(* CODESYS project PETO.export

Project tree, tasks and I/O mapping:
  Device : CODESYS Control Win V3 x64, CODESYS, version 3.5.21.40
    application Application
      libraries: Standard, 3.5.18.0 (System); Util, 3.5.21.0 (System)
      task AlarmManagerTask (cyclic, interval 50 ms, priority 31) calls AlarmManager.Alarm_Prg
      task MainTask (cyclic, interval t#20ms, priority 1) calls COMPROBACION, PREPARACION, SERVIR, SALIDAS
      task VISU_TASK (cyclic, interval 100 ms, priority 31) calls VisuElems.Visu_Prg
      Alarm Configuration
        alarm class Error (priority 10, acknowledge ACK)
        alarm class Info (priority 100, acknowledge REP)
        alarm class Warning (priority 30, acknowledge REP)
        alarm group AlarmGroup
            0 [Error]: Comparison Equal, ExpressionToCompare TRUE, Expression PREPARACION.ErrC - "Falla en el calentador"
            1 [Error]: Comparison Equal, ExpressionToCompare TRUE, Expression PREPARACION.ErrM - "Falla del motor mezclador"
        AlarmStorage
        text list AlarmGroup
      program COMPROBACION [LD]
      visualisation Visualization
  program PREPARACION [LD]
  program SALIDAS [LD]
  program SERVIR [LD]
*)

// Device/Application/COMPROBACION
PROGRAM COMPROBACION
VAR
	START: BOOL;
	STOP: BOOL;
	Inicio: BOOL;
	VO: BOOL;
	Current_State: INT := 10;
	State_machine: INT := 10;
	P1: BOOL;
	L1: BOOL;
	Q1: BOOL;
	RE: BOOL;
	D: BOOL;
	aux1: BOOL;
	V: BOOL;
	aux2: BOOL;
END_VAR
VAR // added by the converter: edge detectors and wires of the graphical bodies
    _w1, _w2, _w3 : BOOL;
END_VAR

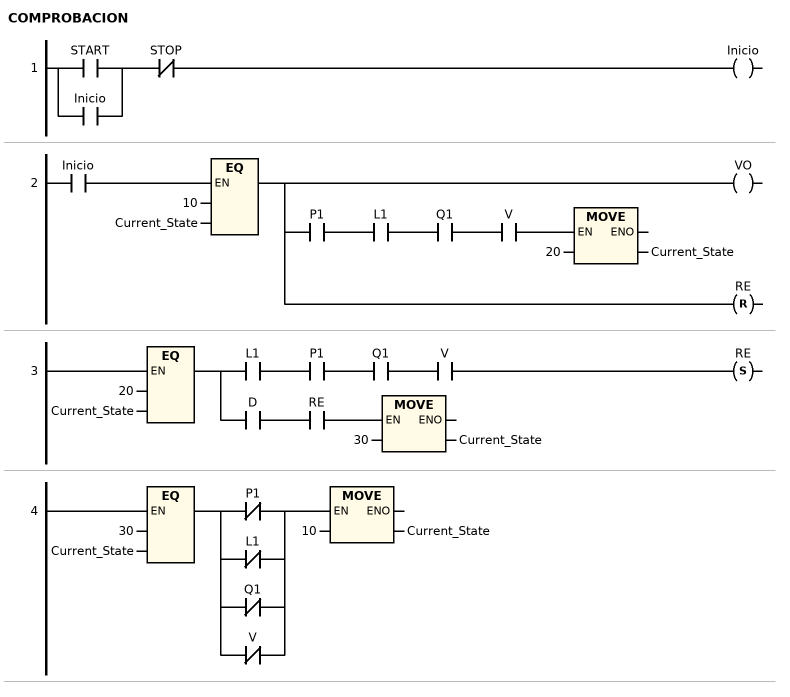
// NETWORK 1
Inicio := (START OR Inicio) AND NOT STOP;

// NETWORK 2
_w1 := Inicio AND 10 = Current_State;
VO := _w1;
IF _w1 AND P1 AND L1 AND Q1 AND V THEN Current_State := 20; END_IF
RE R= _w1;

// NETWORK 3
_w2 := 20 = Current_State;
RE S= _w2 AND L1 AND P1 AND Q1 AND V;
IF _w2 AND D AND RE THEN Current_State := 30; END_IF

// NETWORK 4
_w3 := 30 = Current_State;
IF _w3 AND (NOT P1 OR NOT L1 OR NOT Q1 OR NOT V) THEN Current_State := 10; END_IF

END_PROGRAM

// PREPARACION
PROGRAM PREPARACION
VAR
	RE: BOOL;
	aux1: BOOL;
	CCurrent_State: INT := 10;
	P2: BOOL;
	M1: BOOL;
	// Calentadaor
	K1: BOOL;
	// motor principal
	MO: BOOL;
	TIMERPETO: TON;
	// el tiempo de espera se cumplio
	Tim1: BOOL;
	// error de calentador
	ErrC: BOOL;
	// temperatura tanque
	H1: INT;
	// MANTENIMIENTO
	Mt: BOOL;
	// error de motor
	ErrM: BOOL;
	TIMERMOTOR: TON;
	// peto listo
	Ro: BOOL;
END_VAR
VAR // added by the converter: edge detectors and wires of the graphical bodies
    _w1, _w2, _w3, _w4 : BOOL;
END_VAR

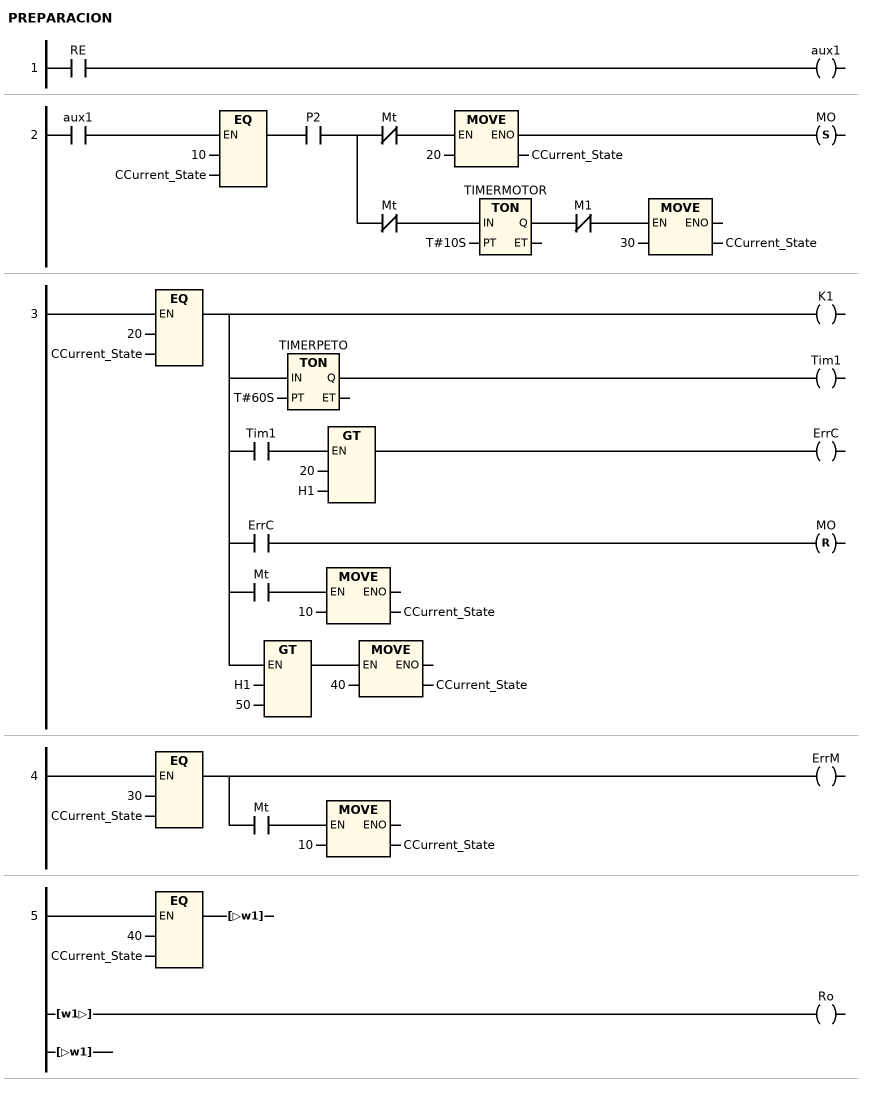
// NETWORK 1
aux1 := RE;

// NETWORK 2
_w1 := (aux1 AND 10 = CCurrent_State) AND P2;
IF _w1 AND NOT Mt THEN CCurrent_State := 20; END_IF
MO S= _w1 AND NOT Mt;
TIMERMOTOR(IN := _w1 AND NOT Mt, PT := T#10S); // TON
IF TIMERMOTOR.Q AND NOT M1 THEN CCurrent_State := 30; END_IF

// NETWORK 3
_w2 := 20 = CCurrent_State;
K1 := _w2;
TIMERPETO(IN := _w2, PT := T#60S); // TON
Tim1 := TIMERPETO.Q;
ErrC := _w2 AND Tim1 AND 20 > H1;
MO R= _w2 AND ErrC;
IF _w2 AND Mt THEN CCurrent_State := 10; END_IF
IF _w2 AND H1 > 50 THEN CCurrent_State := 40; END_IF

// NETWORK 4
_w3 := 30 = CCurrent_State;
ErrM := _w3;
IF _w3 AND Mt THEN CCurrent_State := 10; END_IF

// NETWORK 5
_w4 := 40 = CCurrent_State;
Ro := _w4;

END_PROGRAM

// SERVIR
PROGRAM SERVIR
VAR
	RE: BOOL;
	Ro: BOOL;
	CCCurrent_State: INT;
	T1: BOOL;
	T2: BOOL;
	D: BOOL;
	Q2: BOOL;
	timerpeto: TOF;
	// puerta peto
	Pp: BOOL;
	TIMERPETO2: TON;
	timer1: TIME;
	T: SINT;
	aux1: BOOL;
	//Contador de vaso
	V1: BOOL;
	TON_0: TON;
	Mv1: BOOL;
	Q: BOOL;
	Mt: BOOL;
	CT_V1: CTD;
	// PRESENCIA DE VASO
	Vs: BOOL;
	Mv2: BOOL;
	CT_V2: CTD;
	V2: BOOL;
	TON_1: TON;
	TIMERPETO3: TON;
	aux2: BOOL;
	// panela
	P: BOOL;
	// puerta queso
	Pq: BOOL;
	TIMER_QUESO: TON;
	aux3: BOOL;
	// Señal de agregar
	Sn1: BOOL;
	aux4: BOOL;
	TIMER_PANELA: TON;
	aux5: BOOL;
	// puerta panela
	Ppa: BOOL;
	aux6: BOOL;
	aux7: BOOL;
	aux8: BOOL;
	TON_Final: TON;
	// Terminado
	Ff: BOOL;
	// Habilitador
	Hb: BOOL;
	TIMER_PANELA_A: TON;
	TON_1AUX: TON;
	TIMER_QUESO_A: TON;
	TON_2AUX: TON;
END_VAR
VAR // added by the converter: edge detectors and wires of the graphical bodies
    _w1, _w2, _w3, _w4, _w5, _w6, _w7 : BOOL;
END_VAR

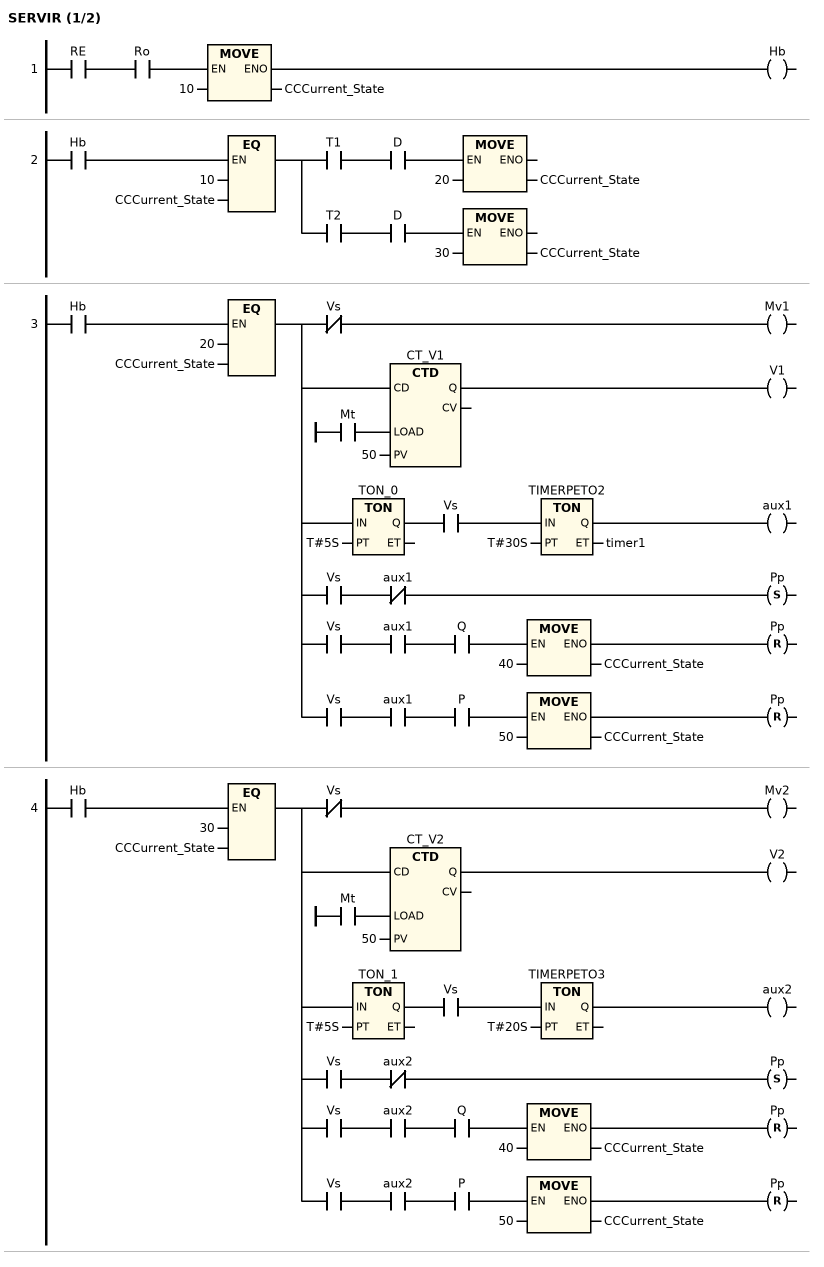
// NETWORK 1
_w1 := RE AND Ro;
IF _w1 THEN CCCurrent_State := 10; END_IF
Hb := _w1;

// NETWORK 2
_w2 := Hb AND 10 = CCCurrent_State;
IF _w2 AND T1 AND D THEN CCCurrent_State := 20; END_IF
IF _w2 AND T2 AND D THEN CCCurrent_State := 30; END_IF

// NETWORK 3
_w3 := Hb AND 20 = CCCurrent_State;
Mv1 := _w3 AND NOT Vs;
CT_V1(CD := _w3, LOAD := Mt, PV := 50); // CTD
V1 := CT_V1.Q;
TON_0(IN := _w3, PT := T#5S); // TON
TIMERPETO2(IN := TON_0.Q AND Vs, PT := T#30S, ET => timer1); // TON
aux1 := TIMERPETO2.Q;
Pp S= _w3 AND Vs AND NOT aux1;
IF _w3 AND Vs AND aux1 AND Q THEN CCCurrent_State := 40; END_IF
Pp R= _w3 AND Vs AND aux1 AND Q;
IF _w3 AND Vs AND aux1 AND P THEN CCCurrent_State := 50; END_IF
Pp R= _w3 AND Vs AND aux1 AND P;

// NETWORK 4
_w4 := Hb AND 30 = CCCurrent_State;
Mv2 := _w4 AND NOT Vs;
CT_V2(CD := _w4, LOAD := Mt, PV := 50); // CTD
V2 := CT_V2.Q;
TON_1(IN := _w4, PT := T#5S); // TON
TIMERPETO3(IN := TON_1.Q AND Vs, PT := T#20S); // TON
aux2 := TIMERPETO3.Q;
Pp S= _w4 AND Vs AND NOT aux2;
IF _w4 AND Vs AND aux2 AND Q THEN CCCurrent_State := 40; END_IF
Pp R= _w4 AND Vs AND aux2 AND Q;
IF _w4 AND Vs AND aux2 AND P THEN CCCurrent_State := 50; END_IF
Pp R= _w4 AND Vs AND aux2 AND P;

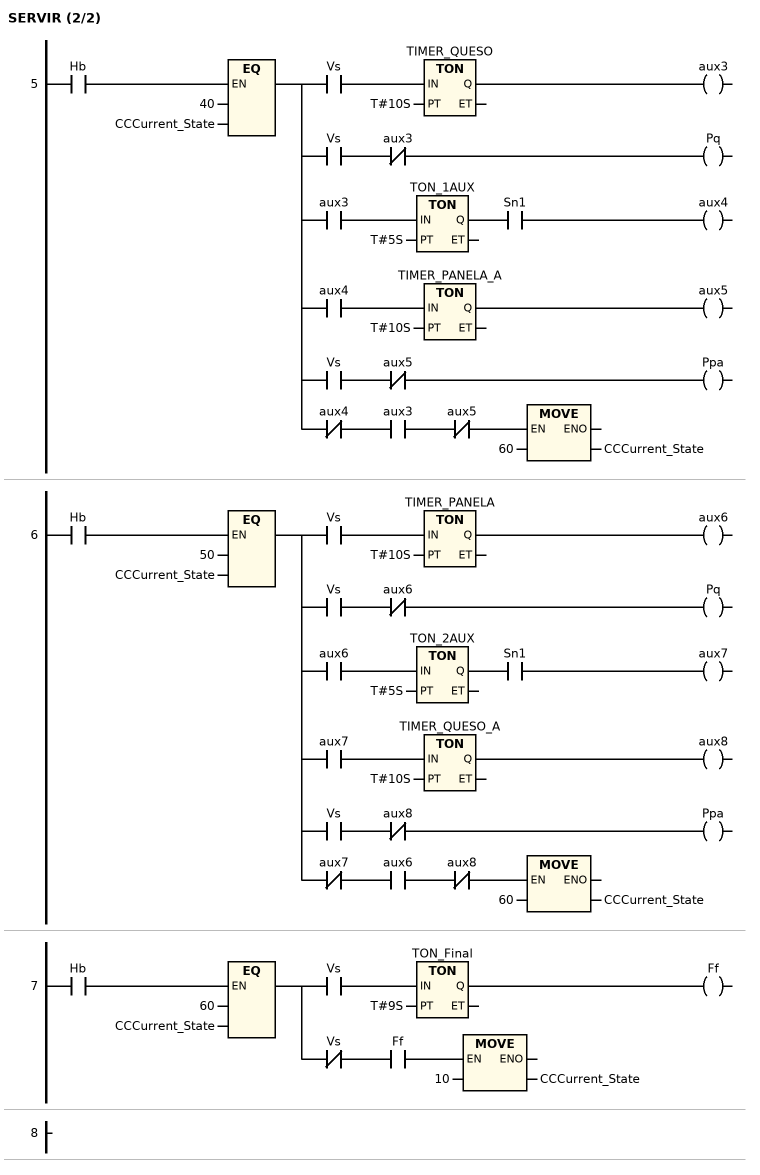
// NETWORK 5
_w5 := Hb AND 40 = CCCurrent_State;
TIMER_QUESO(IN := _w5 AND Vs, PT := T#10S); // TON
aux3 := TIMER_QUESO.Q;
Pq := _w5 AND Vs AND NOT aux3;
TON_1AUX(IN := _w5 AND aux3, PT := T#5S); // TON
aux4 := TON_1AUX.Q AND Sn1;
TIMER_PANELA_A(IN := _w5 AND aux4, PT := T#10S); // TON
aux5 := TIMER_PANELA_A.Q;
Ppa := _w5 AND Vs AND NOT aux5;
IF _w5 AND NOT aux4 AND aux3 AND NOT aux5 THEN CCCurrent_State := 60; END_IF

// NETWORK 6
_w6 := Hb AND 50 = CCCurrent_State;
TIMER_PANELA(IN := _w6 AND Vs, PT := T#10S); // TON
aux6 := TIMER_PANELA.Q;
Pq := _w6 AND Vs AND NOT aux6;
TON_2AUX(IN := _w6 AND aux6, PT := T#5S); // TON
aux7 := TON_2AUX.Q AND Sn1;
TIMER_QUESO_A(IN := _w6 AND aux7, PT := T#10S); // TON
aux8 := TIMER_QUESO_A.Q;
Ppa := _w6 AND Vs AND NOT aux8;
IF _w6 AND NOT aux7 AND aux6 AND NOT aux8 THEN CCCurrent_State := 60; END_IF

// NETWORK 7
_w7 := Hb AND 60 = CCCurrent_State;
TON_Final(IN := _w7 AND Vs, PT := T#9S); // TON
Ff := TON_Final.Q;
IF _w7 AND NOT Vs AND Ff THEN CCCurrent_State := 10; END_IF

// NETWORK 8

END_PROGRAM

// SALIDAS
PROGRAM SALIDAS
VAR
	MO: BOOL;
	// erro calentaddor
	ErrC: BOOL;
	// salida del motor
	O1: BOOL;
	// error motor
	ErrM: BOOL;
	K1: BOOL;
	// salida del calentador
	O2: BOOL;
END_VAR

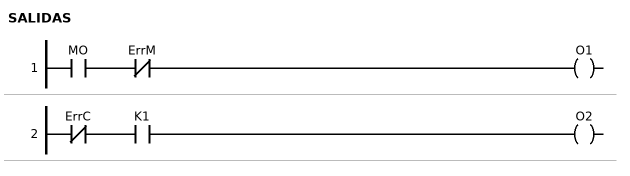
// NETWORK 1
O1 := MO AND NOT ErrM;

// NETWORK 2
O2 := NOT ErrC AND K1;

END_PROGRAM

// Device/Application/Visualization
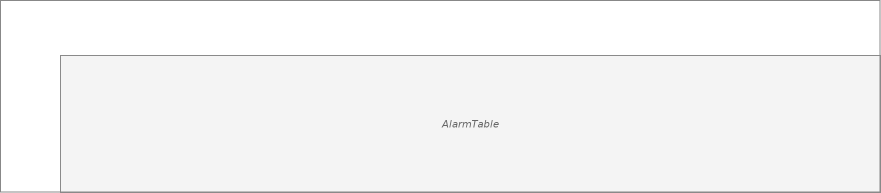
VISUALIZATION Visualization  // 881x193
VAR_IN_OUT
END_VAR
VAR
	bAckSel : BOOL;
	bAckVisible : BOOL;
	bHistory : BOOL;
	bFreezeScrlPos : BOOL;
END_VAR
    AlarmTable (60,55 821x138)
        p1521930926: __All
        p1663851261: __All
        p428520879: bAckSel
        p2607059081: bAckVisible
        p3266827225: bHistory
        p3894972949: bFreezeScrlPos
    Button (60,203 90x30), "ACK selected"
        toggle bAckSel
    Button (170,203 90x30), "ACK all visible"
        toggle bAckVisible
    Button (280,203 90x30), "History"
        toggle bHistory
    Button (390,203 90x30), "Freeze Scrl Pos"
        toggle bFreezeScrlPos
END_VISUALIZATION

(* text list AlarmGroup (id | default)
  1 | Falla del motor mezclador
  0 | Falla en el calentador
   |  *)
